# EPICS StreamDevice protocol: source/epics/code/pwmLED/pwmLED.proto
Terminator = CR LF;

putval{
  out "%s";
}
